// TIA Portal V17 export
// export: Created 2026-04-12T10:31:56.5026063Z, ExportSetting WithDefaults, DisplayName Totally Integrated Automation Portal, DisplayVersion V17 Update 4, DisplayName TIA Portal Openness, DisplayVersion V17 Update 4, DisplayName TIA Portal Version Control Interface, DisplayVersion V17, DisplayName SINAMICS Startdrive Advanced, DisplayVersion V17, DisplayName SINAMICS Startdrive G130, G150, S120, S150, SINAMICS MV, S210, DisplayVersion V17, DisplayName SINAMICS Startdrive G110M, G120, G120C, G120D, G120P, G115D, DisplayVersion V17, DisplayName STEP 7 Professional, DisplayVersion V17 Update 4, DisplayName STEP 7 Safety, DisplayVersion V17, DisplayName WinCC Advanced, DisplayVersion V17 Update 4
FUNCTION_BLOCK "程序发生器"   // FB2, LAD
{ S7_Optimized_Access := 'FALSE' }
VERSION : 0.1
// stored: AutoNumber false, IsIECCheckEnabled false, SetENOAutomatically false, UDAEnableTagReadback false
   VAR_INPUT
      程序等待 : Bool;
      初始温度 { ExternalAccessible := 'False'; ExternalVisible := 'False'; ExternalWritable := 'False'} : Real;
      目标温度1 { ExternalAccessible := 'False'; ExternalVisible := 'False'; ExternalWritable := 'False'} : Real;
      目标温度2 { ExternalAccessible := 'False'; ExternalVisible := 'False'; ExternalWritable := 'False'} : Real;
      目标温度3 { ExternalAccessible := 'False'; ExternalVisible := 'False'; ExternalWritable := 'False'} : Real;
      目标温度4 { ExternalAccessible := 'False'; ExternalVisible := 'False'; ExternalWritable := 'False'} : Real;
      目标温度5 { ExternalAccessible := 'False'; ExternalVisible := 'False'; ExternalWritable := 'False'} : Real;
      升温斜率1 : Real;
      升温斜率2 : Real;
      升温斜率3 : Real;
      升温斜率4 : Real;
      升温斜率5 : Real;
      保温时间1 { ExternalAccessible := 'False'; ExternalVisible := 'False'; ExternalWritable := 'False'} : Real;
      保温时间2 { ExternalAccessible := 'False'; ExternalVisible := 'False'; ExternalWritable := 'False'} : Real;
      保温时间3 { ExternalAccessible := 'False'; ExternalVisible := 'False'; ExternalWritable := 'False'} : Real;
      保温时间4 { ExternalAccessible := 'False'; ExternalVisible := 'False'; ExternalWritable := 'False'} : Real;
      保温时间5 { ExternalAccessible := 'False'; ExternalVisible := 'False'; ExternalWritable := 'False'} : Real;
   END_VAR
   VAR_OUTPUT
      设定值 : Real;
      当前段数 { ExternalAccessible := 'False'; ExternalVisible := 'False'; ExternalWritable := 'False'} : Int;
      当前段剩余时间分钟 { ExternalAccessible := 'False'; ExternalVisible := 'False'; ExternalWritable := 'False'} : Real;
      总剩余时间 { ExternalAccessible := 'False'; ExternalVisible := 'False'; ExternalWritable := 'False'} : Real;
      程序运行标识 { ExternalAccessible := 'False'; ExternalVisible := 'False'; ExternalWritable := 'False'} : Bool;
      程序升温标识 { ExternalAccessible := 'False'; ExternalVisible := 'False'; ExternalWritable := 'False'} : Bool;
      程序降温标识 { ExternalAccessible := 'False'; ExternalVisible := 'False'; ExternalWritable := 'False'} : Bool;
      程序保温标识 { ExternalAccessible := 'False'; ExternalVisible := 'False'; ExternalWritable := 'False'} : Bool;
      "总运行时间小时（含暂停）" { ExternalAccessible := 'False'; ExternalVisible := 'False'; ExternalWritable := 'False'} : Real;
      运行时间小时 { ExternalAccessible := 'False'; ExternalVisible := 'False'; ExternalWritable := 'False'} : Real;
      "总运行时间分（含暂停）" { ExternalAccessible := 'False'; ExternalVisible := 'False'; ExternalWritable := 'False'} : Real;
      运行时间分 { ExternalAccessible := 'False'; ExternalVisible := 'False'; ExternalWritable := 'False'} : Real;
      升温时间1 { ExternalAccessible := 'False'; ExternalVisible := 'False'; ExternalWritable := 'False'} : Real;
      升温时间2 { ExternalAccessible := 'False'; ExternalVisible := 'False'; ExternalWritable := 'False'} : Real;
      升温时间3 { ExternalAccessible := 'False'; ExternalVisible := 'False'; ExternalWritable := 'False'} : Real;
      升温时间4 { ExternalAccessible := 'False'; ExternalVisible := 'False'; ExternalWritable := 'False'} : Real;
      升温时间5 { ExternalAccessible := 'False'; ExternalVisible := 'False'; ExternalWritable := 'False'} : Real;
      时间和10 { ExternalAccessible := 'False'; ExternalVisible := 'False'; ExternalWritable := 'False'} : Real;
      当前剩余时间小时 : Real;
   END_VAR
   VAR_IN_OUT
      运行 : Bool;
      暂停 : Bool;
      曲线发送 : Bool;
      跳步 : Bool;
   END_VAR
   VAR DB_SPECIFIC
      时间和1 { ExternalAccessible := 'False'; ExternalVisible := 'False'; ExternalWritable := 'False'} : Real;
      时间和2 { ExternalAccessible := 'False'; ExternalVisible := 'False'; ExternalWritable := 'False'} : Real;
      时间和3 { ExternalAccessible := 'False'; ExternalVisible := 'False'; ExternalWritable := 'False'} : Real;
      时间和4 { ExternalAccessible := 'False'; ExternalVisible := 'False'; ExternalWritable := 'False'} : Real;
      时间和5 { ExternalAccessible := 'False'; ExternalVisible := 'False'; ExternalWritable := 'False'} : Real;
      时间和6 { ExternalAccessible := 'False'; ExternalVisible := 'False'; ExternalWritable := 'False'} : Real;
      时间和7 { ExternalAccessible := 'False'; ExternalVisible := 'False'; ExternalWritable := 'False'} : Real;
      时间和8 { ExternalAccessible := 'False'; ExternalVisible := 'False'; ExternalWritable := 'False'} : Real;
      时间和9 { ExternalAccessible := 'False'; ExternalVisible := 'False'; ExternalWritable := 'False'} : Real;
      运行时间秒 { ExternalAccessible := 'False'; ExternalVisible := 'False'; ExternalWritable := 'False'} : Int;
      "总运行时间秒（含暂停）" { ExternalAccessible := 'False'; ExternalVisible := 'False'; ExternalWritable := 'False'} : Real;
      过程温度1 { ExternalAccessible := 'False'; ExternalVisible := 'False'; ExternalWritable := 'False'} : Real;
      过程温度2 { ExternalAccessible := 'False'; ExternalVisible := 'False'; ExternalWritable := 'False'} : Real;
      过程时间分钟 { ExternalAccessible := 'False'; ExternalVisible := 'False'; ExternalWritable := 'False'} : Real;
      过程差值 { ExternalAccessible := 'False'; ExternalVisible := 'False'; ExternalWritable := 'False'} : Real;
      过程时间秒 { ExternalAccessible := 'False'; ExternalVisible := 'False'; ExternalWritable := 'False'} : Real;
      商 { ExternalAccessible := 'False'; ExternalVisible := 'False'; ExternalWritable := 'False'} : Real;
      程序发送脉冲 { ExternalAccessible := 'False'; ExternalVisible := 'False'; ExternalWritable := 'False'} : Bool;
      程序运行脉冲 { ExternalAccessible := 'False'; ExternalVisible := 'False'; ExternalWritable := 'False'} : Bool;
      程序跳步脉冲 { ExternalAccessible := 'False'; ExternalVisible := 'False'; ExternalWritable := 'False'} : Bool;
      秒脉冲 { ExternalAccessible := 'False'; ExternalVisible := 'False'; ExternalWritable := 'False'} : Bool;
      程序运行脉冲1 : Bool;
      程序停止脉冲1 : Bool;
      程序停止脉冲2 : Bool;
      程序停止脉冲3 : Bool;
      曲线延时定时器 : IEC_TIMER;
      程序跳步定时器 { S7_SetPoint := 'True'} : IEC_TIMER;
   END_VAR
   VAR_TEMP   // added for the SCL form of the ladder/FBD networks
      _w1 : Bool;
      _w2 : Bool;
      _w3 : Bool;
      _w4 : Bool;
      _w5 : Bool;
      _w6 : Bool;
   END_VAR
BEGIN

REGION Network 1: 升温时间计算
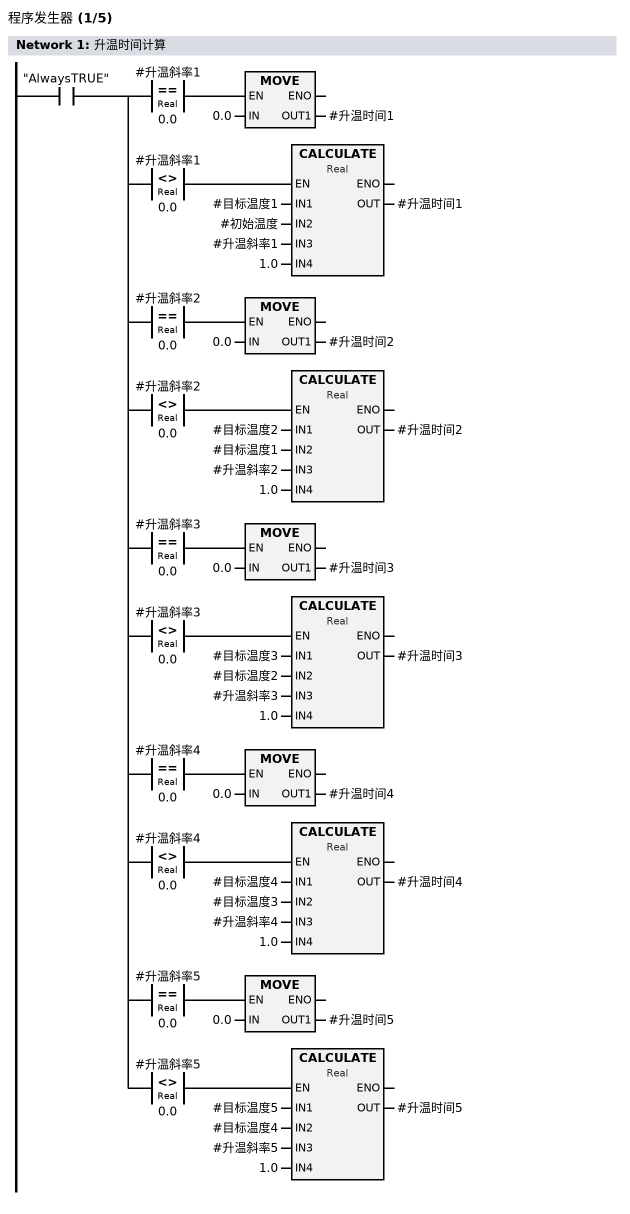
   RUNG wire#powerrail
      Contact( "AlwaysTRUE" )
      wire#w1
      { S7_Templates := "SrcType := Real" } EQ_Contact(in1 := #升温斜率1, in2 := 0.0)
      Move(in := 0.0, out1 => #升温时间1)
   END_RUNG
   RUNG wire#w1
      { S7_Templates := "SrcType := Real" } NE_Contact(in1 := #升温斜率1, in2 := 0.0)
      { S7_Templates := "SrcType := Real"; S7_Expression := "(ABS(IN1-IN2)/IN3)*IN4" } Calculate(in1 := #目标温度1, in2 := #初始温度, in3 := #升温斜率1, in4 := 1.0, out => #升温时间1)
   END_RUNG
   RUNG wire#w1
      { S7_Templates := "SrcType := Real" } EQ_Contact(in1 := #升温斜率2, in2 := 0.0)
      Move(in := 0.0, out1 => #升温时间2)
   END_RUNG
   RUNG wire#w1
      { S7_Templates := "SrcType := Real" } NE_Contact(in1 := #升温斜率2, in2 := 0.0)
      { S7_Templates := "SrcType := Real"; S7_Expression := "(ABS(IN1-IN2)/IN3)*IN4" } Calculate(in1 := #目标温度2, in2 := #目标温度1, in3 := #升温斜率2, in4 := 1.0, out => #升温时间2)
   END_RUNG
   RUNG wire#w1
      { S7_Templates := "SrcType := Real" } EQ_Contact(in1 := #升温斜率3, in2 := 0.0)
      Move(in := 0.0, out1 => #升温时间3)
   END_RUNG
   RUNG wire#w1
      { S7_Templates := "SrcType := Real" } NE_Contact(in1 := #升温斜率3, in2 := 0.0)
      { S7_Templates := "SrcType := Real"; S7_Expression := "(ABS(IN1-IN2)/IN3)*IN4" } Calculate(in1 := #目标温度3, in2 := #目标温度2, in3 := #升温斜率3, in4 := 1.0, out => #升温时间3)
   END_RUNG
   RUNG wire#w1
      { S7_Templates := "SrcType := Real" } EQ_Contact(in1 := #升温斜率4, in2 := 0.0)
      Move(in := 0.0, out1 => #升温时间4)
   END_RUNG
   RUNG wire#w1
      { S7_Templates := "SrcType := Real" } NE_Contact(in1 := #升温斜率4, in2 := 0.0)
      { S7_Templates := "SrcType := Real"; S7_Expression := "(ABS(IN1-IN2)/IN3)*IN4" } Calculate(in1 := #目标温度4, in2 := #目标温度3, in3 := #升温斜率4, in4 := 1.0, out => #升温时间4)
   END_RUNG
   RUNG wire#w1
      { S7_Templates := "SrcType := Real" } EQ_Contact(in1 := #升温斜率5, in2 := 0.0)
      Move(in := 0.0, out1 => #升温时间5)
   END_RUNG
   RUNG wire#w1
      { S7_Templates := "SrcType := Real" } NE_Contact(in1 := #升温斜率5, in2 := 0.0)
      { S7_Templates := "SrcType := Real"; S7_Expression := "(ABS(IN1-IN2)/IN3)*IN4" } Calculate(in1 := #目标温度5, in2 := #目标温度4, in3 := #升温斜率5, in4 := 1.0, out => #升温时间5)
   END_RUNG
   // the same network as SCL:
   IF "AlwaysTRUE" AND (#升温斜率1 = 0.0) THEN #升温时间1 := 0.0; END_IF;
   IF "AlwaysTRUE" AND (#升温斜率1 <> 0.0) THEN #升温时间1 := (ABS(#目标温度1-#初始温度)/#升温斜率1)*1.0; END_IF;
   IF "AlwaysTRUE" AND (#升温斜率2 = 0.0) THEN #升温时间2 := 0.0; END_IF;
   IF "AlwaysTRUE" AND (#升温斜率2 <> 0.0) THEN #升温时间2 := (ABS(#目标温度2-#目标温度1)/#升温斜率2)*1.0; END_IF;
   IF "AlwaysTRUE" AND (#升温斜率3 = 0.0) THEN #升温时间3 := 0.0; END_IF;
   IF "AlwaysTRUE" AND (#升温斜率3 <> 0.0) THEN #升温时间3 := (ABS(#目标温度3-#目标温度2)/#升温斜率3)*1.0; END_IF;
   IF "AlwaysTRUE" AND (#升温斜率4 = 0.0) THEN #升温时间4 := 0.0; END_IF;
   IF "AlwaysTRUE" AND (#升温斜率4 <> 0.0) THEN #升温时间4 := (ABS(#目标温度4-#目标温度3)/#升温斜率4)*1.0; END_IF;
   IF "AlwaysTRUE" AND (#升温斜率5 = 0.0) THEN #升温时间5 := 0.0; END_IF;
   IF "AlwaysTRUE" AND (#升温斜率5 <> 0.0) THEN #升温时间5 := (ABS(#目标温度5-#目标温度4)/#升温斜率5)*1.0; END_IF;
END_REGION

REGION Network 2: 时间和统计
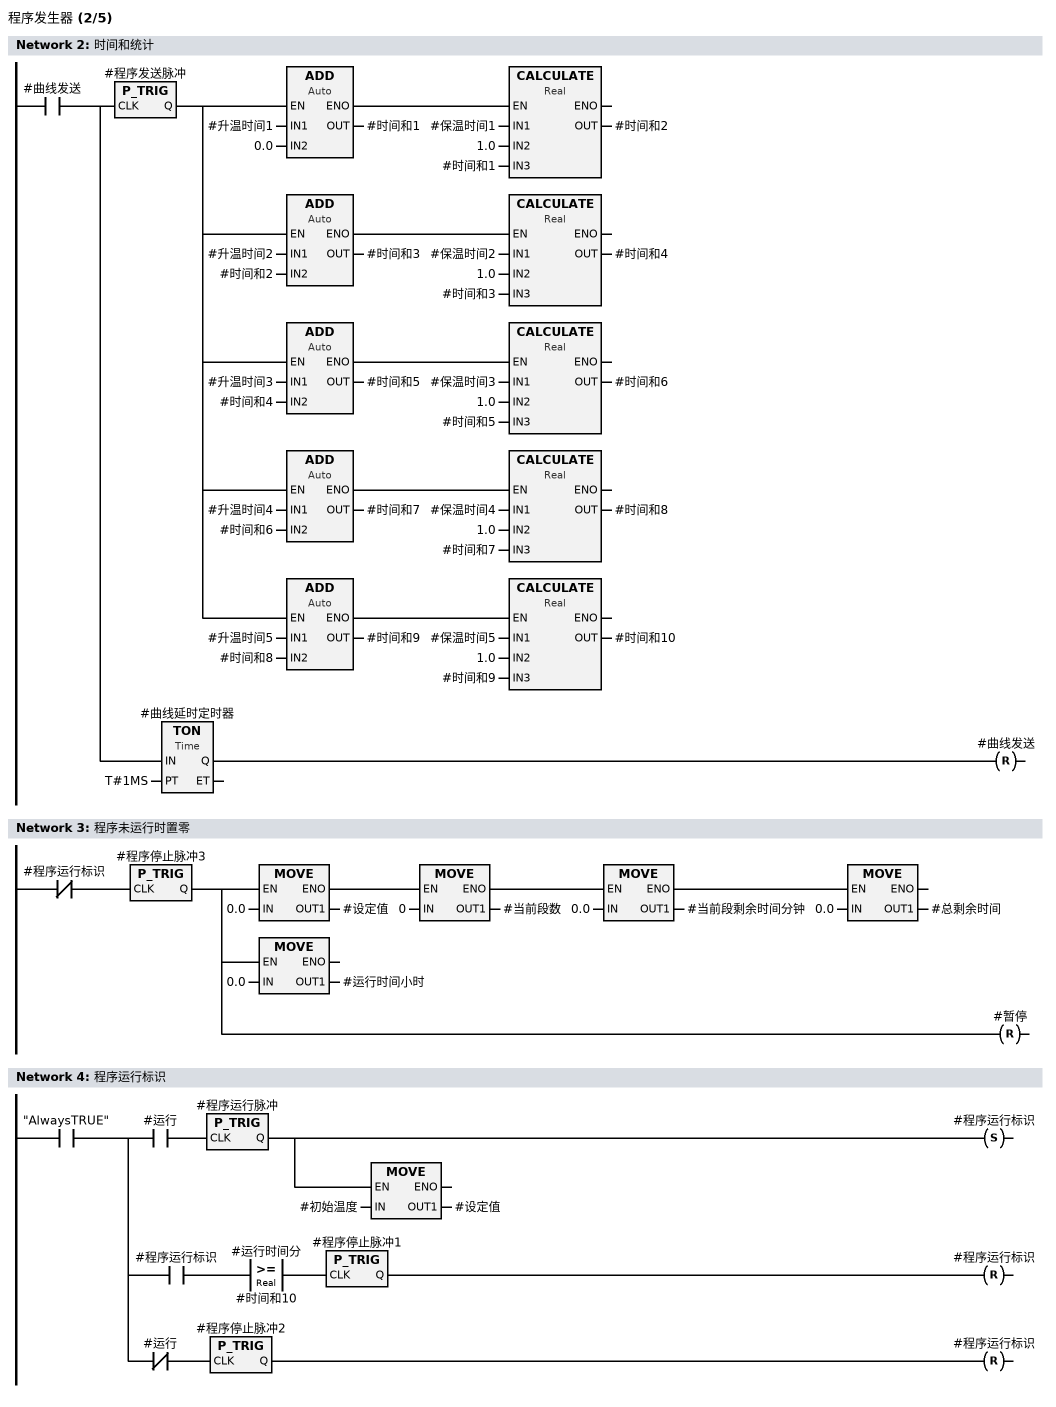
   RUNG wire#powerrail
      Contact( #曲线发送 )
      wire#w1
      P_Trig( #程序发送脉冲 )
      wire#w2
      Add(in1 := #升温时间1, in2 := 0.0, out => #时间和1)
      { S7_Templates := "SrcType := Real"; S7_Expression := "IN1*IN2+IN3" } Calculate(in1 := #保温时间1, in2 := 1.0, in3 := #时间和1, out => #时间和2)
   END_RUNG
   RUNG wire#w2
      Add(in1 := #升温时间2, in2 := #时间和2, out => #时间和3)
      { S7_Templates := "SrcType := Real"; S7_Expression := "IN1*IN2+IN3" } Calculate(in1 := #保温时间2, in2 := 1.0, in3 := #时间和3, out => #时间和4)
   END_RUNG
   RUNG wire#w2
      Add(in1 := #升温时间3, in2 := #时间和4, out => #时间和5)
      { S7_Templates := "SrcType := Real"; S7_Expression := "IN1*IN2+IN3" } Calculate(in1 := #保温时间3, in2 := 1.0, in3 := #时间和5, out => #时间和6)
   END_RUNG
   RUNG wire#w2
      Add(in1 := #升温时间4, in2 := #时间和6, out => #时间和7)
      { S7_Templates := "SrcType := Real"; S7_Expression := "IN1*IN2+IN3" } Calculate(in1 := #保温时间4, in2 := 1.0, in3 := #时间和7, out => #时间和8)
   END_RUNG
   RUNG wire#w2
      Add(in1 := #升温时间5, in2 := #时间和8, out => #时间和9)
      { S7_Templates := "SrcType := Real"; S7_Expression := "IN1*IN2+IN3" } Calculate(in1 := #保温时间5, in2 := 1.0, in3 := #时间和9, out => #时间和10)
   END_RUNG
   RUNG wire#w1
      { S7_Templates := "time_type := Time" } #曲线延时定时器.TON(pt := T#1MS, et =>)
      R_Coil( #曲线发送 )
   END_RUNG
   // the same network as SCL:
   #_w1 := #曲线发送 AND NOT #程序发送脉冲;   // rising edge
   #程序发送脉冲 := #曲线发送;
   IF #_w1 THEN
       #时间和1 := #升温时间1 + 0.0;
       #时间和2 := #保温时间1*1.0+#时间和1;
       #时间和3 := #升温时间2 + #时间和2;
       #时间和4 := #保温时间2*1.0+#时间和3;
       #时间和5 := #升温时间3 + #时间和4;
       #时间和6 := #保温时间3*1.0+#时间和5;
       #时间和7 := #升温时间4 + #时间和6;
       #时间和8 := #保温时间4*1.0+#时间和7;
       #时间和9 := #升温时间5 + #时间和8;
       #时间和10 := #保温时间5*1.0+#时间和9;
   END_IF;
   #曲线延时定时器.TON(IN := #曲线发送, PT := T#1MS);
   IF #曲线延时定时器.Q THEN #曲线发送 := FALSE; END_IF;
END_REGION

REGION Network 3: 程序未运行时置零
   RUNG wire#powerrail
      I_Contact( #程序运行标识 )
      P_Trig( #程序停止脉冲3 )
      wire#w1
      Move(in := 0.0, out1 => #设定值)
      Move(in := 0, out1 => #当前段数)
      Move(in := 0.0, out1 => #当前段剩余时间分钟)
      Move(in := 0.0, out1 => #总剩余时间)
   END_RUNG
   RUNG wire#w1
      Move(in := 0.0, out1 => #运行时间小时)
   END_RUNG
   RUNG wire#w1
      R_Coil( #暂停 )
   END_RUNG
   // the same network as SCL:
   #_w1 := NOT #程序运行标识 AND NOT #程序停止脉冲3;   // rising edge
   #程序停止脉冲3 := NOT #程序运行标识;
   IF #_w1 THEN
       #设定值 := 0.0;
       #当前段数 := 0;
       #当前段剩余时间分钟 := 0.0;
       #总剩余时间 := 0.0;
       #运行时间小时 := 0.0;
       #暂停 := FALSE;
   END_IF;
END_REGION

REGION Network 4: 程序运行标识
   RUNG wire#powerrail
      Contact( "AlwaysTRUE" )
      wire#w1
      Contact( #运行 )
      P_Trig( #程序运行脉冲 )
      wire#w2
      S_Coil( #程序运行标识 )
   END_RUNG
   RUNG wire#w2
      Move(in := #初始温度, out1 => #设定值)
   END_RUNG
   RUNG wire#w1
      Contact( #程序运行标识 )
      { S7_Templates := "SrcType := Real" } GE_Contact(in1 := #运行时间分, in2 := #时间和10)
      P_Trig( #程序停止脉冲1 )
      R_Coil( #程序运行标识 )
   END_RUNG
   RUNG wire#w1
      I_Contact( #运行 )
      P_Trig( #程序停止脉冲2 )
      R_Coil( #程序运行标识 )
   END_RUNG
   // the same network as SCL:
   #_w1 := "AlwaysTRUE" AND #运行;
   #_w2 := #_w1 AND NOT #程序运行脉冲;   // rising edge
   #程序运行脉冲 := #_w1;
   IF #_w2 THEN
       #程序运行标识 := TRUE;
       #设定值 := #初始温度;
   END_IF;
   #_w3 := "AlwaysTRUE" AND #程序运行标识 AND (#运行时间分 >= #时间和10);
   #_w4 := #_w3 AND NOT #程序停止脉冲1;   // rising edge
   #程序停止脉冲1 := #_w3;
   IF #_w4 THEN #程序运行标识 := FALSE; END_IF;
   #_w5 := "AlwaysTRUE" AND NOT #运行;
   #_w6 := #_w5 AND NOT #程序停止脉冲2;   // rising edge
   #程序停止脉冲2 := #_w5;
   IF #_w6 THEN #程序运行标识 := FALSE; END_IF;
END_REGION

REGION Network 5: 程序计时及跳步、设定温度变化
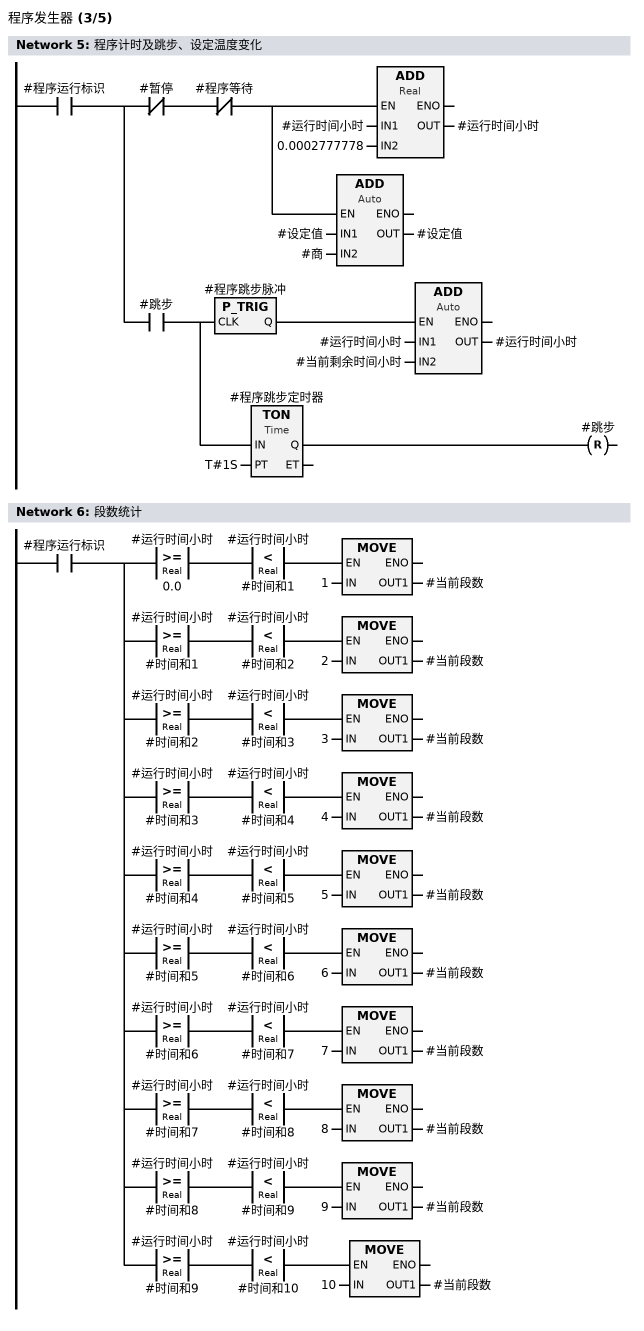
   RUNG wire#powerrail
      Contact( #程序运行标识 )
      wire#w1
      I_Contact( #暂停 )
      I_Contact( #程序等待 )
      wire#w2
      { S7_Templates := "SrcType := Real" } Add(in1 := #运行时间小时, in2 := 0.0002777778, out => #运行时间小时)
   END_RUNG
   RUNG wire#w2
      Add(in1 := #设定值, in2 := #商, out => #设定值)
   END_RUNG
   RUNG wire#w1
      Contact( #跳步 )
      wire#w3
      P_Trig( #程序跳步脉冲 )
      Add(in1 := #运行时间小时, in2 := #当前剩余时间小时, out => #运行时间小时)
   END_RUNG
   RUNG wire#w3
      { S7_Templates := "time_type := Time" } #程序跳步定时器.TON(pt := T#1S, et =>)
      R_Coil( #跳步 )
   END_RUNG
   // the same network as SCL:
   IF #程序运行标识 AND NOT #暂停 AND NOT #程序等待 THEN
       #运行时间小时 := #运行时间小时 + 0.0002777778;
       #设定值 := #设定值 + #商;
   END_IF;
   #_w1 := #程序运行标识 AND #跳步;
   #_w2 := #_w1 AND NOT #程序跳步脉冲;   // rising edge
   #程序跳步脉冲 := #_w1;
   IF #_w2 THEN #运行时间小时 := #运行时间小时 + #当前剩余时间小时; END_IF;
   #程序跳步定时器.TON(IN := #_w1, PT := T#1S);
   IF #程序跳步定时器.Q THEN #跳步 := FALSE; END_IF;
END_REGION

REGION Network 6: 段数统计
   RUNG wire#powerrail
      Contact( #程序运行标识 )
      wire#w1
      { S7_Templates := "SrcType := Real" } GE_Contact(in1 := #运行时间小时, in2 := 0.0)
      { S7_Templates := "SrcType := Real" } LT_Contact(in1 := #运行时间小时, in2 := #时间和1)
      Move(in := 1, out1 => #当前段数)
   END_RUNG
   RUNG wire#w1
      { S7_Templates := "SrcType := Real" } GE_Contact(in1 := #运行时间小时, in2 := #时间和1)
      { S7_Templates := "SrcType := Real" } LT_Contact(in1 := #运行时间小时, in2 := #时间和2)
      Move(in := 2, out1 => #当前段数)
   END_RUNG
   RUNG wire#w1
      { S7_Templates := "SrcType := Real" } GE_Contact(in1 := #运行时间小时, in2 := #时间和2)
      { S7_Templates := "SrcType := Real" } LT_Contact(in1 := #运行时间小时, in2 := #时间和3)
      Move(in := 3, out1 => #当前段数)
   END_RUNG
   RUNG wire#w1
      { S7_Templates := "SrcType := Real" } GE_Contact(in1 := #运行时间小时, in2 := #时间和3)
      { S7_Templates := "SrcType := Real" } LT_Contact(in1 := #运行时间小时, in2 := #时间和4)
      Move(in := 4, out1 => #当前段数)
   END_RUNG
   RUNG wire#w1
      { S7_Templates := "SrcType := Real" } GE_Contact(in1 := #运行时间小时, in2 := #时间和4)
      { S7_Templates := "SrcType := Real" } LT_Contact(in1 := #运行时间小时, in2 := #时间和5)
      Move(in := 5, out1 => #当前段数)
   END_RUNG
   RUNG wire#w1
      { S7_Templates := "SrcType := Real" } GE_Contact(in1 := #运行时间小时, in2 := #时间和5)
      { S7_Templates := "SrcType := Real" } LT_Contact(in1 := #运行时间小时, in2 := #时间和6)
      Move(in := 6, out1 => #当前段数)
   END_RUNG
   RUNG wire#w1
      { S7_Templates := "SrcType := Real" } GE_Contact(in1 := #运行时间小时, in2 := #时间和6)
      { S7_Templates := "SrcType := Real" } LT_Contact(in1 := #运行时间小时, in2 := #时间和7)
      Move(in := 7, out1 => #当前段数)
   END_RUNG
   RUNG wire#w1
      { S7_Templates := "SrcType := Real" } GE_Contact(in1 := #运行时间小时, in2 := #时间和7)
      { S7_Templates := "SrcType := Real" } LT_Contact(in1 := #运行时间小时, in2 := #时间和8)
      Move(in := 8, out1 => #当前段数)
   END_RUNG
   RUNG wire#w1
      { S7_Templates := "SrcType := Real" } GE_Contact(in1 := #运行时间小时, in2 := #时间和8)
      { S7_Templates := "SrcType := Real" } LT_Contact(in1 := #运行时间小时, in2 := #时间和9)
      Move(in := 9, out1 => #当前段数)
   END_RUNG
   RUNG wire#w1
      { S7_Templates := "SrcType := Real" } GE_Contact(in1 := #运行时间小时, in2 := #时间和9)
      { S7_Templates := "SrcType := Real" } LT_Contact(in1 := #运行时间小时, in2 := #时间和10)
      Move(in := 10, out1 => #当前段数)
   END_RUNG
   // the same network as SCL:
   IF #程序运行标识 AND (#运行时间小时 >= 0.0) AND (#运行时间小时 < #时间和1) THEN #当前段数 := 1; END_IF;
   IF #程序运行标识 AND (#运行时间小时 >= #时间和1) AND (#运行时间小时 < #时间和2) THEN #当前段数 := 2; END_IF;
   IF #程序运行标识 AND (#运行时间小时 >= #时间和2) AND (#运行时间小时 < #时间和3) THEN #当前段数 := 3; END_IF;
   IF #程序运行标识 AND (#运行时间小时 >= #时间和3) AND (#运行时间小时 < #时间和4) THEN #当前段数 := 4; END_IF;
   IF #程序运行标识 AND (#运行时间小时 >= #时间和4) AND (#运行时间小时 < #时间和5) THEN #当前段数 := 5; END_IF;
   IF #程序运行标识 AND (#运行时间小时 >= #时间和5) AND (#运行时间小时 < #时间和6) THEN #当前段数 := 6; END_IF;
   IF #程序运行标识 AND (#运行时间小时 >= #时间和6) AND (#运行时间小时 < #时间和7) THEN #当前段数 := 7; END_IF;
   IF #程序运行标识 AND (#运行时间小时 >= #时间和7) AND (#运行时间小时 < #时间和8) THEN #当前段数 := 8; END_IF;
   IF #程序运行标识 AND (#运行时间小时 >= #时间和8) AND (#运行时间小时 < #时间和9) THEN #当前段数 := 9; END_IF;
   IF #程序运行标识 AND (#运行时间小时 >= #时间和9) AND (#运行时间小时 < #时间和10) THEN #当前段数 := 10; END_IF;
END_REGION

REGION Network 7: 当前段温度、时间过渡及当前段剩余时间计算
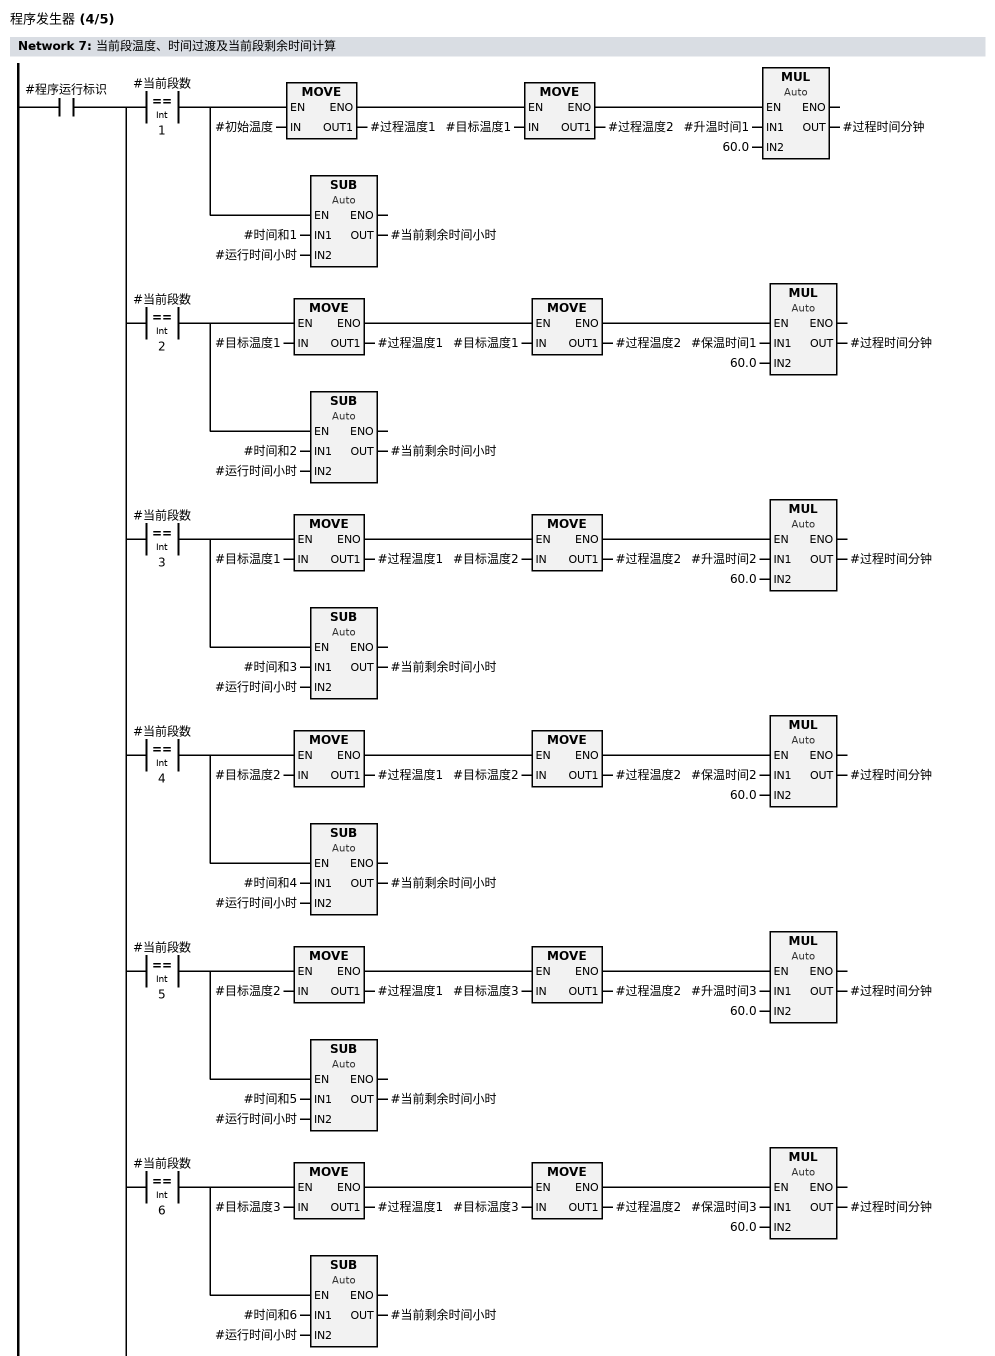
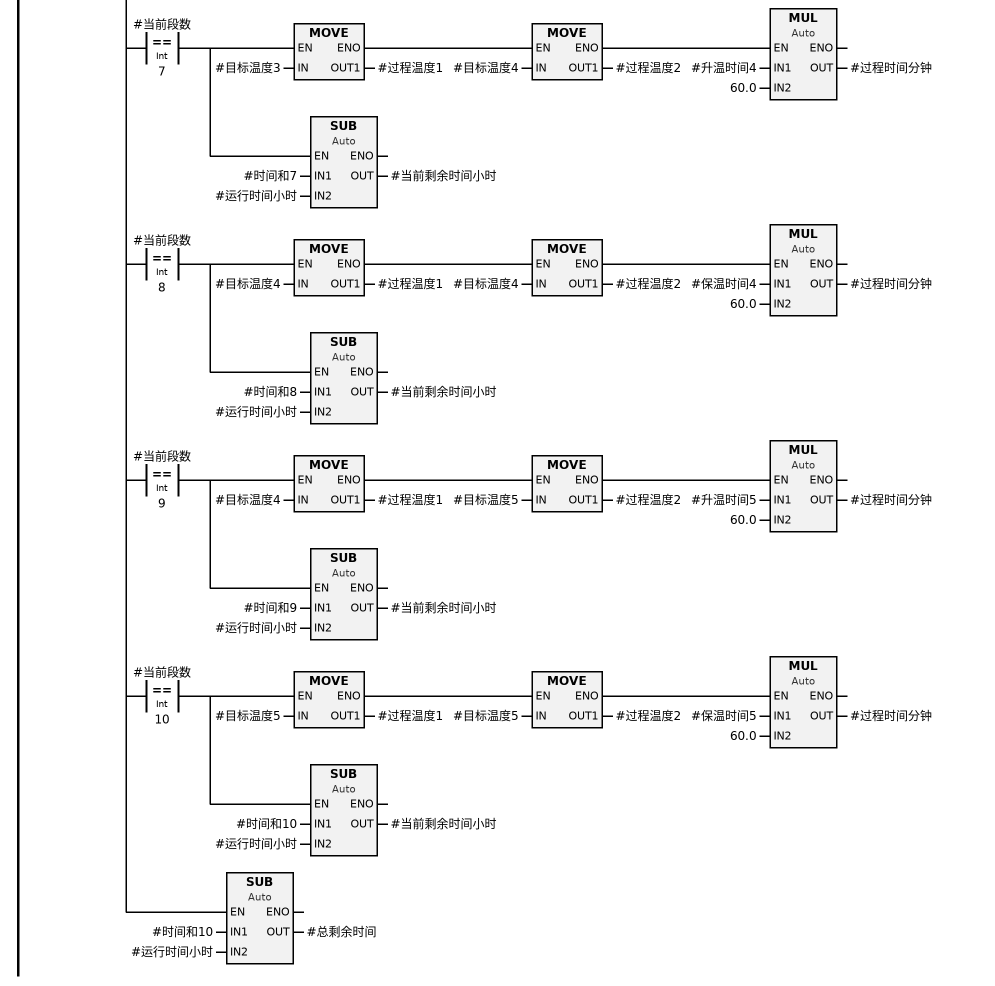
   RUNG wire#powerrail
      Contact( #程序运行标识 )
      wire#w1
      { S7_Templates := "SrcType := Int" } EQ_Contact(in1 := #当前段数, in2 := 1)
      wire#w2
      Move(in := #初始温度, out1 => #过程温度1)
      Move(in := #目标温度1, out1 => #过程温度2)
      Mul(in1 := #升温时间1, in2 := 60.0, out => #过程时间分钟)
   END_RUNG
   RUNG wire#w2
      Sub(in1 := #时间和1, in2 := #运行时间小时, out => #当前剩余时间小时)
   END_RUNG
   RUNG wire#w1
      { S7_Templates := "SrcType := Int" } EQ_Contact(in1 := #当前段数, in2 := 2)
      wire#w3
      Move(in := #目标温度1, out1 => #过程温度1)
      Move(in := #目标温度1, out1 => #过程温度2)
      Mul(in1 := #保温时间1, in2 := 60.0, out => #过程时间分钟)
   END_RUNG
   RUNG wire#w3
      Sub(in1 := #时间和2, in2 := #运行时间小时, out => #当前剩余时间小时)
   END_RUNG
   RUNG wire#w1
      { S7_Templates := "SrcType := Int" } EQ_Contact(in1 := #当前段数, in2 := 3)
      wire#w4
      Move(in := #目标温度1, out1 => #过程温度1)
      Move(in := #目标温度2, out1 => #过程温度2)
      Mul(in1 := #升温时间2, in2 := 60.0, out => #过程时间分钟)
   END_RUNG
   RUNG wire#w4
      Sub(in1 := #时间和3, in2 := #运行时间小时, out => #当前剩余时间小时)
   END_RUNG
   RUNG wire#w1
      { S7_Templates := "SrcType := Int" } EQ_Contact(in1 := #当前段数, in2 := 4)
      wire#w5
      Move(in := #目标温度2, out1 => #过程温度1)
      Move(in := #目标温度2, out1 => #过程温度2)
      Mul(in1 := #保温时间2, in2 := 60.0, out => #过程时间分钟)
   END_RUNG
   RUNG wire#w5
      Sub(in1 := #时间和4, in2 := #运行时间小时, out => #当前剩余时间小时)
   END_RUNG
   RUNG wire#w1
      { S7_Templates := "SrcType := Int" } EQ_Contact(in1 := #当前段数, in2 := 5)
      wire#w6
      Move(in := #目标温度2, out1 => #过程温度1)
      Move(in := #目标温度3, out1 => #过程温度2)
      Mul(in1 := #升温时间3, in2 := 60.0, out => #过程时间分钟)
   END_RUNG
   RUNG wire#w6
      Sub(in1 := #时间和5, in2 := #运行时间小时, out => #当前剩余时间小时)
   END_RUNG
   RUNG wire#w1
      { S7_Templates := "SrcType := Int" } EQ_Contact(in1 := #当前段数, in2 := 6)
      wire#w7
      Move(in := #目标温度3, out1 => #过程温度1)
      Move(in := #目标温度3, out1 => #过程温度2)
      Mul(in1 := #保温时间3, in2 := 60.0, out => #过程时间分钟)
   END_RUNG
   RUNG wire#w7
      Sub(in1 := #时间和6, in2 := #运行时间小时, out => #当前剩余时间小时)
   END_RUNG
   RUNG wire#w1
      { S7_Templates := "SrcType := Int" } EQ_Contact(in1 := #当前段数, in2 := 7)
      wire#w8
      Move(in := #目标温度3, out1 => #过程温度1)
      Move(in := #目标温度4, out1 => #过程温度2)
      Mul(in1 := #升温时间4, in2 := 60.0, out => #过程时间分钟)
   END_RUNG
   RUNG wire#w8
      Sub(in1 := #时间和7, in2 := #运行时间小时, out => #当前剩余时间小时)
   END_RUNG
   RUNG wire#w1
      { S7_Templates := "SrcType := Int" } EQ_Contact(in1 := #当前段数, in2 := 8)
      wire#w9
      Move(in := #目标温度4, out1 => #过程温度1)
      Move(in := #目标温度4, out1 => #过程温度2)
      Mul(in1 := #保温时间4, in2 := 60.0, out => #过程时间分钟)
   END_RUNG
   RUNG wire#w9
      Sub(in1 := #时间和8, in2 := #运行时间小时, out => #当前剩余时间小时)
   END_RUNG
   RUNG wire#w1
      { S7_Templates := "SrcType := Int" } EQ_Contact(in1 := #当前段数, in2 := 9)
      wire#w10
      Move(in := #目标温度4, out1 => #过程温度1)
      Move(in := #目标温度5, out1 => #过程温度2)
      Mul(in1 := #升温时间5, in2 := 60.0, out => #过程时间分钟)
   END_RUNG
   RUNG wire#w10
      Sub(in1 := #时间和9, in2 := #运行时间小时, out => #当前剩余时间小时)
   END_RUNG
   RUNG wire#w1
      { S7_Templates := "SrcType := Int" } EQ_Contact(in1 := #当前段数, in2 := 10)
      wire#w11
      Move(in := #目标温度5, out1 => #过程温度1)
      Move(in := #目标温度5, out1 => #过程温度2)
      Mul(in1 := #保温时间5, in2 := 60.0, out => #过程时间分钟)
   END_RUNG
   RUNG wire#w11
      Sub(in1 := #时间和10, in2 := #运行时间小时, out => #当前剩余时间小时)
   END_RUNG
   RUNG wire#w1
      Sub(in1 := #时间和10, in2 := #运行时间小时, out => #总剩余时间)
   END_RUNG
   // the same network as SCL:
   IF #程序运行标识 AND (#当前段数 = 1) THEN
       #过程温度1 := #初始温度;
       #过程温度2 := #目标温度1;
       #过程时间分钟 := #升温时间1 * 60.0;
       #当前剩余时间小时 := #时间和1 - #运行时间小时;
   END_IF;
   IF #程序运行标识 AND (#当前段数 = 2) THEN
       #过程温度1 := #目标温度1;
       #过程温度2 := #目标温度1;
       #过程时间分钟 := #保温时间1 * 60.0;
       #当前剩余时间小时 := #时间和2 - #运行时间小时;
   END_IF;
   IF #程序运行标识 AND (#当前段数 = 3) THEN
       #过程温度1 := #目标温度1;
       #过程温度2 := #目标温度2;
       #过程时间分钟 := #升温时间2 * 60.0;
       #当前剩余时间小时 := #时间和3 - #运行时间小时;
   END_IF;
   IF #程序运行标识 AND (#当前段数 = 4) THEN
       #过程温度1 := #目标温度2;
       #过程温度2 := #目标温度2;
       #过程时间分钟 := #保温时间2 * 60.0;
       #当前剩余时间小时 := #时间和4 - #运行时间小时;
   END_IF;
   IF #程序运行标识 AND (#当前段数 = 5) THEN
       #过程温度1 := #目标温度2;
       #过程温度2 := #目标温度3;
       #过程时间分钟 := #升温时间3 * 60.0;
       #当前剩余时间小时 := #时间和5 - #运行时间小时;
   END_IF;
   IF #程序运行标识 AND (#当前段数 = 6) THEN
       #过程温度1 := #目标温度3;
       #过程温度2 := #目标温度3;
       #过程时间分钟 := #保温时间3 * 60.0;
       #当前剩余时间小时 := #时间和6 - #运行时间小时;
   END_IF;
   IF #程序运行标识 AND (#当前段数 = 7) THEN
       #过程温度1 := #目标温度3;
       #过程温度2 := #目标温度4;
       #过程时间分钟 := #升温时间4 * 60.0;
       #当前剩余时间小时 := #时间和7 - #运行时间小时;
   END_IF;
   IF #程序运行标识 AND (#当前段数 = 8) THEN
       #过程温度1 := #目标温度4;
       #过程温度2 := #目标温度4;
       #过程时间分钟 := #保温时间4 * 60.0;
       #当前剩余时间小时 := #时间和8 - #运行时间小时;
   END_IF;
   IF #程序运行标识 AND (#当前段数 = 9) THEN
       #过程温度1 := #目标温度4;
       #过程温度2 := #目标温度5;
       #过程时间分钟 := #升温时间5 * 60.0;
       #当前剩余时间小时 := #时间和9 - #运行时间小时;
   END_IF;
   IF #程序运行标识 AND (#当前段数 = 10) THEN
       #过程温度1 := #目标温度5;
       #过程温度2 := #目标温度5;
       #过程时间分钟 := #保温时间5 * 60.0;
       #当前剩余时间小时 := #时间和10 - #运行时间小时;
   END_IF;
   IF #程序运行标识 THEN #总剩余时间 := #时间和10 - #运行时间小时; END_IF;
END_REGION

REGION Network 8: 商计算
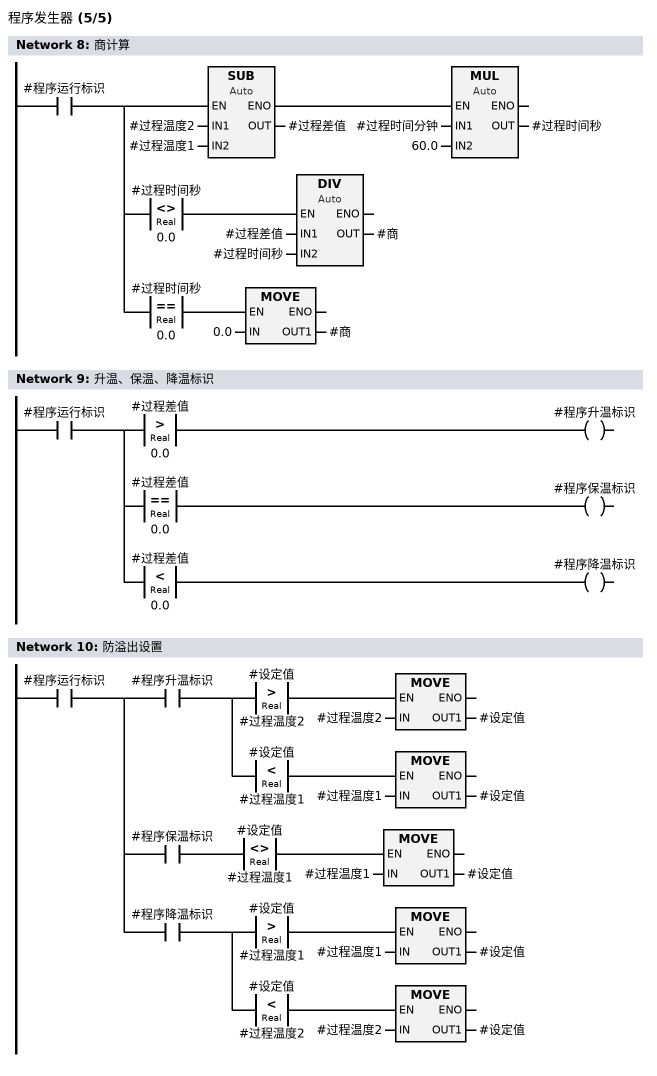
   RUNG wire#powerrail
      Contact( #程序运行标识 )
      wire#w1
      Sub(in1 := #过程温度2, in2 := #过程温度1, out => #过程差值)
      Mul(in1 := #过程时间分钟, in2 := 60.0, out => #过程时间秒)
   END_RUNG
   RUNG wire#w1
      { S7_Templates := "SrcType := Real" } NE_Contact(in1 := #过程时间秒, in2 := 0.0)
      Div(in1 := #过程差值, in2 := #过程时间秒, out => #商)
   END_RUNG
   RUNG wire#w1
      { S7_Templates := "SrcType := Real" } EQ_Contact(in1 := #过程时间秒, in2 := 0.0)
      Move(in := 0.0, out1 => #商)
   END_RUNG
   // the same network as SCL:
   IF #程序运行标识 THEN
       #过程差值 := #过程温度2 - #过程温度1;
       #过程时间秒 := #过程时间分钟 * 60.0;
   END_IF;
   IF #程序运行标识 AND (#过程时间秒 <> 0.0) THEN #商 := #过程差值 / #过程时间秒; END_IF;
   IF #程序运行标识 AND (#过程时间秒 = 0.0) THEN #商 := 0.0; END_IF;
END_REGION

REGION Network 9: 升温、保温、降温标识
   RUNG wire#powerrail
      Contact( #程序运行标识 )
      wire#w1
      { S7_Templates := "SrcType := Real" } GT_Contact(in1 := #过程差值, in2 := 0.0)
      Coil( #程序升温标识 )
   END_RUNG
   RUNG wire#w1
      { S7_Templates := "SrcType := Real" } EQ_Contact(in1 := #过程差值, in2 := 0.0)
      Coil( #程序保温标识 )
   END_RUNG
   RUNG wire#w1
      { S7_Templates := "SrcType := Real" } LT_Contact(in1 := #过程差值, in2 := 0.0)
      Coil( #程序降温标识 )
   END_RUNG
   // the same network as SCL:
   #程序升温标识 := #程序运行标识 AND (#过程差值 > 0.0);
   #程序保温标识 := #程序运行标识 AND (#过程差值 = 0.0);
   #程序降温标识 := #程序运行标识 AND (#过程差值 < 0.0);
END_REGION

REGION Network 10: 防溢出设置
   RUNG wire#powerrail
      Contact( #程序运行标识 )
      wire#w1
      Contact( #程序升温标识 )
      wire#w2
      { S7_Templates := "SrcType := Real" } GT_Contact(in1 := #设定值, in2 := #过程温度2)
      Move(in := #过程温度2, out1 => #设定值)
   END_RUNG
   RUNG wire#w2
      { S7_Templates := "SrcType := Real" } LT_Contact(in1 := #设定值, in2 := #过程温度1)
      Move(in := #过程温度1, out1 => #设定值)
   END_RUNG
   RUNG wire#w1
      Contact( #程序保温标识 )
      { S7_Templates := "SrcType := Real" } NE_Contact(in1 := #设定值, in2 := #过程温度1)
      Move(in := #过程温度1, out1 => #设定值)
   END_RUNG
   RUNG wire#w1
      Contact( #程序降温标识 )
      wire#w3
      { S7_Templates := "SrcType := Real" } GT_Contact(in1 := #设定值, in2 := #过程温度1)
      Move(in := #过程温度1, out1 => #设定值)
   END_RUNG
   RUNG wire#w3
      { S7_Templates := "SrcType := Real" } LT_Contact(in1 := #设定值, in2 := #过程温度2)
      Move(in := #过程温度2, out1 => #设定值)
   END_RUNG
   // the same network as SCL:
   #_w1 := #程序运行标识 AND #程序升温标识;
   IF #_w1 AND (#设定值 > #过程温度2) THEN #设定值 := #过程温度2; END_IF;
   IF #_w1 AND (#设定值 < #过程温度1) THEN #设定值 := #过程温度1; END_IF;
   IF #程序运行标识 AND #程序保温标识 AND (#设定值 <> #过程温度1) THEN #设定值 := #过程温度1; END_IF;
   #_w2 := #程序运行标识 AND #程序降温标识;
   IF #_w2 AND (#设定值 > #过程温度1) THEN #设定值 := #过程温度1; END_IF;
   IF #_w2 AND (#设定值 < #过程温度2) THEN #设定值 := #过程温度2; END_IF;
END_REGION
END_FUNCTION_BLOCK
